PROGRAM P_EjectionGate
VAR
		(*Initialization*)
	bEJ_OK		: BOOL;
	bError		: BOOL;
	bStart		: BOOL;
	bStop		: BOOL;
	(*Process*)
	bEjEnable 	: BOOL;
	bEjectOn	: BOOL;
	bEjectOff	: BOOL;
	bOverride	: BOOL;
	(*Ejection Gate Specific Process*)
	bSheetStuck		: BOOL;
	bSheetPresence		: BOOL;
	nSheetCount		: INT;
	FB_SheetCount_Trig	: R_TRIG;
	tSheetStuck_s	: TIME :=T#5S ;
	
	
	//-----------------------------------------(*Case*)-----------------------------------------------------
	
	(* Reference for VBT

	State_Init 					,
	State_AutoStart         	,
	State_AutoStop          	,
	State_AutoEjectOn			,
	State_AutoBackToInit        ,
	State_Override				,
	State_Error			
	*)	
	
	asd: R_TRIG;
	FbSheetStuckCheck: TON;
END_VAR
VAR_INPUT
	bStartCommand : BOOL;
END_VAR
VAR_OUTPUT
	iEJcase : INT;
END_VAR

CASE iEJcase OF
EjectionGateState.State_Init			:	

	IF (bEJ_OK AND bStartCommand)  
	AND NOT bError THEN
		iEJcase:= EjectionGateState.State_AutoStart;
	END_IF 
	IF bError THEN
		iEJcase:= EjectionGateState.State_Error;
	END_IF

   
EjectionGateState.State_AutoStart     	:
	IF bStop THEN
		iEJcase:= EjectionGateState.State_AutoStop;
	ELSE
		iEJcase :=EjectionGateState.State_AutoEjectOn;
	END_IF


EjectionGateState.State_AutoStop      	:
	iEJcase:= EjectionGateState.State_AutoBackToInit;


EjectionGateState.State_AutoEjectOn	  	:
	(*Insert business logic here*)
	(*Ejection*)
	IF P_VacummBeltTable.bBadSheetSignal THEN
		bEjectOn :=TRUE;
	END_IF // Need to add business logic to count for speed/time on-site.
	
	(*Sheet Counting*)
	FB_SheetCount_Trig(CLK:= bSheetPresence, Q=> );
	IF FB_SheetCount_Trig.Q THEN
		nSheetCount:=nSheetCount+1;
	END_IF
	FbSheetStuckCheck(IN:=bSheetPresence , PT:=tSheetStuck_s , Q=> , ET=> );
	IF FbSheetStuckCheck.Q THEN
		bSheetStuck:=TRUE;
		iEJcase:= EjectionGateState.State_Error;
	END_IF


EjectionGateState.State_AutoBackToInit	:
	iEJcase:= EjectionGateState.State_Init;


EjectionGateState.State_Override		:   
	;


EjectionGateState.State_Error			:     
	IF bError THEN
		iEJcase:= EjectionGateState.State_AutoBackToInit;
	END_IF

END_CASE

END_PROGRAM

(* stored: Version 1.1.0.1, ProductVersion 3.1.4024.12
   POU P_EjectionGate: Id {6064b460-bcdf-4343-8336-f08ee00714f6}, SpecialFunc None *)
